RoboDK station: welding operation.rdk

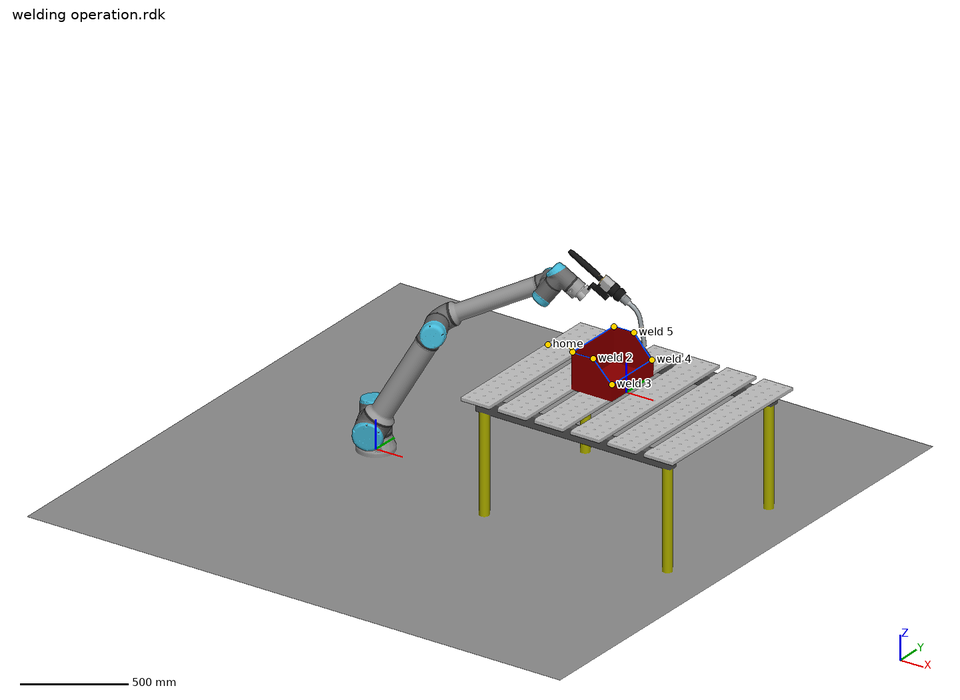
[picture v0: the station drawn from its stored meshes, robots at their saved joint values, targets as dots, program paths as lines]
Station welding operation (saved by RoboDK 6.1.1). Poses are relative to the parent item; angles as X-Y-Z fixed-axis rotations.
  - object Floor at (0, 0, 0) mm, size 3000 x 3000 x 0 mm, geometry from Floor.sld
  - frame Frame 1 at (734.49, 128.3, 611.58) mm
    - object Table 1200x1000mm (Welding) at (0, 0, 0) mm, size 1193.8 x 965.2 x 609.6 mm, geometry from Table-1200x1000mm-Welding.sld
    - object Bin Red at (0, -120, 0) mm, size 225 x 337.5 x 191.2 mm, geometry from Bin-Red.sld
    - target home (Cartesian target) at (-233.55, -298.87, 299.57) mm, rotated rx -180 ry 45 rz -180 deg; joints [9.246, 45.856, -96.32, -129.537, 80.754, 90] of UR10e
    - target weld 1 (Cartesian target) at (-221.56, -116.63, 191.25) mm, rotated rx 169.08 ry 2.09 rz -169.29 deg; joints [7.82, 27.391, -102.492, -147.586, 99.832, 95.79] of UR10e
    - target weld 2 (Cartesian target) at (-106.11, -116.87, 191.18) mm, rotated rx 165.25 ry 2.76 rz -169.46 deg; joints [-130.273, -210.003, 113.486, -40.103, 250.878, 126.727] of UR10e
    - target weld 3 (Cartesian target) at (-3.13, -113.43, 82.4) mm, rotated rx -177.94 ry 10.83 rz -169.17 deg; joints [-134.882, -108.428, -128.474, 96.889, 240.853, 109.778] of UR10e
    - target weld 4 (Cartesian target) at (-3.38, 210.15, 82.44) mm, rotated rx -177.94 ry 10.83 rz -169.17 deg; joints [-41.324, 23.505, -137.774, 67.502, 230.383, 233.41] of UR10e
    - target weld 5 (Cartesian target) at (-107.49, 213.58, 191.11) mm, rotated rx 165.38 ry 3.4 rz -167.17 deg; joints [-26.636, 8.212, -126.743, 64.36, 232.253, 248.869] of UR10e
    - target weld 6 (Cartesian target) at (-220.9, 213.93, 191.2) mm, rotated rx 165.74 ry 3.32 rz -167.16 deg; joints [-21.496, 28.382, -107.757, -151.81, 124.367, 73.681] of UR10e
    - target approace weld (Cartesian target) at (-222.57, -122.66, 219.99) mm, rotated rx 169.08 ry 2.09 rz -169.29 deg; joints [2.9, -107.444, -37.622, -78.311, 103.43, 92.363] of UR10e
  - frame UR10e Base at (-588.94, 3.58, 0) mm
    - robot UR10e: 6 axes, payload 10 kg, reach 1300 mm, repeatability 0.05 mm, weight 28.9 kg
        modified DH rows (alpha deg, a mm, theta deg, d mm): 0, 0, 0, 180.7; 90, 0, 180, 0; 0, 612.6, 0, 0; 0, 571.335, 0, 174.15; -90, 0, 0, 119.85; 90, 0, 180, 116.55
        joint limits [-360, -360, -360, -360, -360, -360] to [360, 360, 360, 360, 360, 360]; home [0, -90, -90, 0, 90, 0]; saved at [25.618, -119.569, -35.912, -61.828, 81.403, 101.473]
      - tool OTC Daihen FD-84 Welding Gun, TCP at (2, 0, 402) mm, rotated rx 0 ry 45 rz 0 deg, size 201.6 x 65.1 x 567.7 mm
  - program Prog1 (12 instructions, listed below)
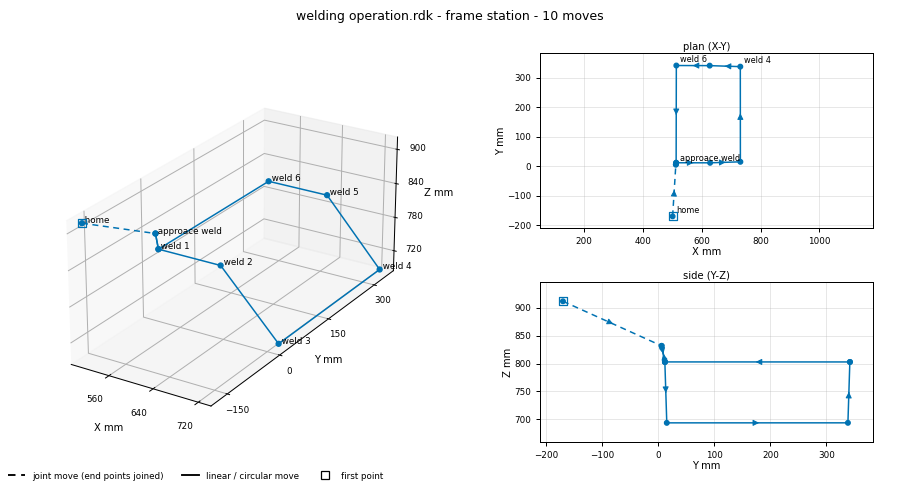
[picture p0: tool path of welding operation.rdk in frame station, 10 of 10 moves have a stored position in this frame; points joined in program order, loops and branches not executed]

--- program Prog1 (robot UR10e) ---
  Set Ref.: Frame 1
  Set Tool: OTC Daihen FD-84 Welding Gun
  MoveJ (home)
  MoveJ (approace weld)
  MoveL (weld 1)
  MoveL (weld 2)
  MoveL (weld 3)
  MoveL (weld 4)
  MoveL (weld 5)
  MoveL (weld 6)
  MoveL (weld 1)
  MoveL (approace weld)
